PROGRAM MAIN
VAR
	//Linking variables to IO cards
	Flow_Valve_1 AT %Q* : INT;
	Level_Valve_1 AT %Q* : INT;
	Level_Valve_2 AT %Q* : INT;
	Level_Valve_3 AT %Q* : INT;
	Gas_Valve AT %Q* : INT;
	Mixer_Valve AT %Q* : INT;
	Motor_speed AT %Q* : INT;
	Motor_ON_OFF AT %Q* :BOOL;
	Motor_Direction AT %Q* :BOOL; 
	Start_Button AT %I* :BOOL;
	Stop_Button AT %I* : BOOL; 
	EMERGENCY_STOP AT %I* : BOOL; 
	Level_Transmitter_1 AT %I* :INT; 
	Level_Transmitter_2 AT %I* :INT; 
	Temperature_Transmitter AT %I* :INT;  
	Pressure_Differencial_Transmitter_1 AT %I* : INT;
	Pressure_Differencial_Transmitter_2 AT %I* : INT;
	Pressure_Transmitter_1 AT %I* : INT ; 
	Pressure_Transmitter_2 AT %I* : INT ; 
	Pressure_Transmitter_3 AT %I* : INT ; 

	
	//User Input as percentage
	Flow_Valve_1_Percentage: INT :=100;
	Level_Valve_1_Percentage: INT    ;
	Level_Valve_2_Percentage: INT;
	Level_Valve_3_Percentage: INT;
	Motor_speed_Percentage: INT; 
	Motor_ON : BOOL ; 
	ON_OFF : STRING(10) := 'OFF' ; 
	
	
	
	
END_VAR



// variable interval for Flow_Valve_1_Percentage  form 0 to 100  
IF Flow_Valve_1_Percentage > 100 THEN
	Flow_Valve_1_Percentage := 100; 
	ELSE IF Flow_Valve_1_Percentage < 0 THEN 
		Flow_Valve_1_Percentage := 0; 
	END_IF
	
END_IF

// variable interval for Level_Valve_1_Percentage  form 0 to 100  
IF Level_Valve_1_Percentage > 100 THEN
	Level_Valve_1_Percentage := 100; 
	ELSE IF Level_Valve_1_Percentage < 0 THEN 
		Level_Valve_1_Percentage := 0; 
	END_IF
	
END_IF

// variable interval for Level_Valve_2_Percentage  form 0 to 100 
IF Level_Valve_2_Percentage > 100 THEN
	Level_Valve_2_Percentage := 100; 
	ELSE IF Level_Valve_2_Percentage < 0 THEN 
		Level_Valve_2_Percentage := 0; 
	END_IF
	
END_IF

// variable interval for Level_Valve_3_Percentage  form 0 to 100 
IF Level_Valve_3_Percentage > 100 THEN
	Level_Valve_3_Percentage := 100; 
	ELSE IF Level_Valve_3_Percentage < 0 THEN 
		Level_Valve_3_Percentage := 0; 
	END_IF
	
END_IF



// variable interval for Motor_speed_Percentage  form 0 to 100 
IF Motor_speed_Percentage > 100 THEN
	Motor_speed_Percentage := 100; 
	ELSE IF Motor_speed_Percentage < 0 THEN 
		Motor_speed_Percentage := 0; 
	END_IF
	
END_IF

// Flow_Valve_1 calibration
Flow_Valve_1 := REAL_TO_INT (262.14*Flow_Valve_1_Percentage +6553 ); 

// Level_Valve_1 calibration
Level_Valve_1 := REAL_TO_INT(262.14*Level_Valve_1_Percentage +6553);

// Level_Valve_2 calibration
Level_Valve_2 := REAL_TO_INT(262.14*Level_Valve_2_Percentage +6553);

// Level_Valve_3 calibration
Level_Valve_3 := REAL_TO_INT(262.14*Level_Valve_3_Percentage +6553);


// Motor_speed calibration
Motor_speed := REAL_TO_INT(262.14*Motor_speed_Percentage +6553);

 
IF Motor_ON_OFF   THEN
    Motor_ON   :=  FALSE;
	ON_OFF  := 'MOTOR: ON' ;
	
ELSE
    Motor_ON  := TRUE;
	ON_OFF  := 'MOTOR: OFF' ;
END_IF

END_PROGRAM

(* stored: Version 1.1.0.1, ProductVersion 3.1.4024.12
   POU MAIN: Id {75317203-8f43-4932-aa88-c7b05e9ca563}, SpecialFunc None *)
